// TIA Portal V20 export
FUNCTION_BLOCK "FB_ExtraMissingPart"   // FB76, SCL
{ S7_Optimized_Access := 'TRUE' }
// stored: MemoryReserve 100, SetENOAutomatically false
   VAR
      sRT_UndrilledGripperClosedWithPart : R_TRIG;
      sRT_UndrilledGripperClosedWithoutPart { S7_SetPoint := 'True'} : R_TRIG;
      sRT_DrilledGripperClosedWithPart : R_TRIG;
      sRT_DrilledGripperClosedWithoutPart { S7_SetPoint := 'True'} : R_TRIG;
      sRT_FixturePartControlGood { S7_SetPoint := 'True'} : R_TRIG;
      sRT_FixturePartControlBad { S7_SetPoint := 'True'} : R_TRIG;
      sRT_UndrilledGripperOpen { S7_SetPoint := 'True'} : R_TRIG;
      sRT_DrilledGripperOpen { S7_SetPoint := 'True'} : R_TRIG;
      sTON_UndrilledGripperClosedWithPart { S7_SetPoint := 'True'} : TON_TIME;
      sTON_UndrilledGripperClosedWithoutPart { S7_SetPoint := 'True'} : TON_TIME;
      sTON_DrilledGripperClosedWithPart { S7_SetPoint := 'True'} : TON_TIME;
      sTON_DrilledGripperClosedWithoutPart { S7_SetPoint := 'True'} : TON_TIME;
      sTON_FixturePartControlGood { S7_SetPoint := 'True'} : TON_TIME;
      sTON_FixturePartControlBad { S7_SetPoint := 'True'} : TON_TIME;
      sTON_UndrilledGripperOpen { S7_SetPoint := 'True'} : TON_TIME;
      sTON_DrilledGripperOpen { S7_SetPoint := 'True'} : TON_TIME;
      sExtraPartUndrilledGripper { S7_SetPoint := 'True'} : Bool;
      sExtraPartDrilledGripper : Bool;
      sMissingPartUndrilledGripper { S7_SetPoint := 'True'} : Bool;
      sMissingPartDrilledGripper : Bool;
      sExtraPartFixture : Bool;
      sMissingPartFixture : Bool;
      sGlobalExtraMissing : Bool;
      sUndrilledGripperClosedWithPart : Bool;
      sUndrilledGripperClosedWithoutPart { S7_SetPoint := 'True'} : Bool;
      sDrilledGripperClosedWithPart : Bool;
      sDrilledGripperClosedWithoutPart { S7_SetPoint := 'True'} : Bool;
      sFixturePartControlGood { S7_SetPoint := 'True'} : Bool;
      sFixturePartControlBad { S7_SetPoint := 'True'} : Bool;
      sUndrilledGripperOpen { S7_SetPoint := 'True'} : Bool;
      sDrilledGripperOpen { S7_SetPoint := 'True'} : Bool;
   END_VAR
BEGIN
   REGION Description header 
       //==================================================================================
       // POSALUX Swiss SA / (C) Copyright 2026
       //----------------------------------------------------------------------------------
       // Title: 
       // Comment/Function: 
       // Author: Fabien WALDT
       // Engineering: TIA Portal v20
       //----------------------------------------------------------------------------------
       // Change log table:
       // Version  | Date     | Expert in charge | Changes applied
       // ---------|----------|------------------|-----------------------------------------
       // 00.00.01 | 20260205 | WFA              | First released version
       // =================================================================================
   END_REGION

   REGION Init
       #sExtraPartUndrilledGripper := FALSE;
       #sExtraPartDrilledGripper := FALSE;
       #sMissingPartUndrilledGripper := FALSE;
       #sMissingPartDrilledGripper := FALSE;
       #sExtraPartFixture := FALSE;
       #sMissingPartFixture := FALSE;
   END_REGION

   REGION Inputs Status
       #sTON_UndrilledGripperClosedWithPart(IN := "DB_GestionGripper".sUndrilledGripper.oStateCloseWithPart,
                                            PT := T#100ms);
       #sTON_UndrilledGripperClosedWithoutPart(IN := "DB_GestionGripper".sUndrilledGripper.oStateClose,
                                               PT := T#100ms);
       #sTON_DrilledGripperClosedWithPart(IN := "DB_GestionGripper".sDrilledGripper.oStateCloseWithPart,
                                          PT := T#100ms);
       #sTON_DrilledGripperClosedWithoutPart(IN := "DB_GestionGripper".sDrilledGripper.oStateClose,
                                             PT := T#100ms);
       #sTON_FixturePartControlGood(IN := "DB_GestionFixture".sFixturePartControl.oGoodPart,
                                    PT := T#100ms);
       #sTON_FixturePartControlBad(IN := "DB_GestionFixture".sFixturePartControl.oBadpart,
                                   PT := T#100ms);

       #sTON_UndrilledGripperOpen(IN := "DB_GestionGripper".sUndrilledGripper.oStateOpen,
                                  PT := T#100ms);
       #sTON_DrilledGripperOpen(IN := "DB_GestionGripper".sDrilledGripper.oStateOpen,
                                PT := T#100ms);

       #sRT_UndrilledGripperClosedWithPart(CLK := #sTON_UndrilledGripperClosedWithPart.Q);
       #sRT_UndrilledGripperClosedWithoutPart(CLK := #sTON_UndrilledGripperClosedWithoutPart.Q);
       #sRT_DrilledGripperClosedWithPart(CLK := #sTON_DrilledGripperClosedWithPart.Q);
       #sRT_DrilledGripperClosedWithoutPart(CLK := #sTON_DrilledGripperClosedWithoutPart.Q);
       #sRT_FixturePartControlGood(CLK := #sTON_FixturePartControlGood.Q);
       #sRT_FixturePartControlBad(CLK := #sTON_FixturePartControlBad.Q);
       #sRT_UndrilledGripperOpen(CLK := #sTON_UndrilledGripperOpen.Q);
       #sRT_DrilledGripperOpen(CLK := #sTON_DrilledGripperOpen.Q);

       #sUndrilledGripperClosedWithPart := #sTON_UndrilledGripperClosedWithPart.Q;
       #sUndrilledGripperClosedWithoutPart := #sTON_UndrilledGripperClosedWithoutPart.Q;
       #sDrilledGripperClosedWithPart := #sTON_DrilledGripperClosedWithPart.Q;
       #sDrilledGripperClosedWithoutPart := #sTON_DrilledGripperClosedWithoutPart.Q;
       #sFixturePartControlGood := #sTON_FixturePartControlGood.Q;
       #sFixturePartControlBad := #sTON_FixturePartControlBad.Q;
       #sUndrilledGripperOpen := #sTON_UndrilledGripperOpen.Q;
       #sDrilledGripperOpen := #sTON_DrilledGripperOpen.Q;

   END_REGION

   REGION Shuttle to Undrilled Gripper
       IF "LBP_ModeGroup".E_JOG THEN
           IF #sRT_UndrilledGripperClosedWithPart.Q AND NOT "DB_PartManagement".sPosition.sGripper.Undrilled.Presence.Part THEN
               "DB_PartManagement".sPosition.sGripper.Undrilled.Presence.Part := TRUE;
               "DB_PartManagement".sPosition.sGripper.Undrilled.Presence.BW := TRUE;
           ELSIF #sRT_UndrilledGripperClosedWithoutPart.Q AND "DB_PartManagement".sPosition.sGripper.Undrilled.Presence.Part THEN
               "DB_PartManagement".sPosition.sGripper.Undrilled.Presence.Part := FALSE;
               "DB_PartManagement".sPosition.sGripper.Undrilled.Presence.BW := FALSE;
           END_IF;
       ELSIF NOT "DB_WorkingModes".sDryRun THEN
           IF #sUndrilledGripperClosedWithPart AND NOT "DB_PartManagement".sPosition.sGripper.Undrilled.Presence.Part THEN
               #sExtraPartUndrilledGripper := TRUE;
               "LBP_AlarmMsgs".UserA[04].A70UUxx[25] := TRUE; // Msg 700425 "Extra Product Undrilled Gripper"
           ELSIF #sUndrilledGripperClosedWithoutPart AND "DB_PartManagement".sPosition.sGripper.Undrilled.Presence.Part THEN
               #sMissingPartUndrilledGripper := TRUE;
               "LBP_AlarmMsgs".UserA[04].A70UUxx[24] := TRUE; // Msg 700424 "Missing Product Undrilled Gripper"
           END_IF;
       END_IF;
   END_REGION

   REGION Undrilled Gripper to Fixture
       IF "LBP_ModeGroup".E_JOG THEN
           IF #sRT_FixturePartControlGood.Q AND NOT "DB_PartManagement".sPosition.sFixture.Undrilled.Presence.Part AND NOT "DB_PartManagement".sPosition.sFixture.Drilled.Presence.Part THEN
               "DB_PartManagement".sPosition.sFixture.Drilled.Presence.Part := TRUE;
               "DB_PartManagement".sPosition.sFixture.Drilled.Presence.BW := TRUE;
           ELSIF #sRT_FixturePartControlBad.Q AND ("DB_PartManagement".sPosition.sFixture.Undrilled.Presence.Part OR "DB_PartManagement".sPosition.sFixture.Drilled.Presence.Part) THEN
               "DB_PartManagement".sPosition.sFixture.Drilled.Presence.Part := FALSE;
               "DB_PartManagement".sPosition.sFixture.Drilled.Presence.BW := FALSE;
           END_IF;
       ELSIF NOT "DB_WorkingModes".sDryRun THEN
           IF #sFixturePartControlGood AND NOT "DB_PartManagement".sPosition.sFixture.Undrilled.Presence.Part AND NOT "DB_PartManagement".sPosition.sFixture.Drilled.Presence.Part THEN
               #sExtraPartFixture := TRUE;
               "LBP_AlarmMsgs".UserA[04].A70UUxx[27] := TRUE; // Msg 700427 "Extra Product Fixture"
           ELSIF #sFixturePartControlBad AND ("DB_PartManagement".sPosition.sFixture.Undrilled.Presence.Part OR "DB_PartManagement".sPosition.sFixture.Drilled.Presence.Part) THEN
               #sMissingPartFixture := TRUE;
               "LBP_AlarmMsgs".UserA[04].A70UUxx[26] := TRUE; // Msg 700426 "Missing Product Fixture"
           END_IF;
       END_IF;
   END_REGION

   REGION Fixture to Drilled Gripper
       IF "LBP_ModeGroup".E_JOG THEN
           IF #sRT_DrilledGripperClosedWithPart.Q AND NOT "DB_PartManagement".sPosition.sGripper.Drilled.Presence.Part THEN
               "DB_PartManagement".sPosition.sGripper.Drilled.Presence.Part := TRUE;
               "DB_PartManagement".sPosition.sGripper.Drilled.Presence.BW := TRUE;
           ELSIF #sRT_DrilledGripperClosedWithoutPart.Q AND "DB_PartManagement".sPosition.sGripper.Drilled.Presence.Part THEN
               "DB_PartManagement".sPosition.sGripper.Drilled.Presence.Part := FALSE;
               "DB_PartManagement".sPosition.sGripper.Drilled.Presence.BW := FALSE;
           END_IF;
       ELSIF NOT "DB_WorkingModes".sDryRun THEN
           IF #sDrilledGripperClosedWithPart AND NOT "DB_PartManagement".sPosition.sGripper.Drilled.Presence.Part THEN
               #sExtraPartDrilledGripper := TRUE;
               "LBP_AlarmMsgs".UserA[04].A70UUxx[29] := TRUE; // Msg 700429 "Extra Product Drilled Gripper"
           ELSIF #sDrilledGripperClosedWithoutPart AND "DB_PartManagement".sPosition.sGripper.Drilled.Presence.Part THEN
               #sMissingPartDrilledGripper := TRUE;
               "LBP_AlarmMsgs".UserA[04].A70UUxx[28] := TRUE; // Msg 700428 "Missing Product Drilled Gripper"
           END_IF;
       END_IF;
   END_REGION

   REGION Gripper Open
       IF "LBP_ModeGroup".E_JOG THEN
           IF #sRT_UndrilledGripperOpen.Q THEN
               "DB_PartManagement".sPosition.sGripper.Undrilled.Presence.Part := FALSE;
               "DB_PartManagement".sPosition.sGripper.Undrilled.Presence.BW := FALSE;
           END_IF;
           IF #sRT_DrilledGripperOpen.Q THEN
               "DB_PartManagement".sPosition.sGripper.Drilled.Presence.Part := FALSE;
               "DB_PartManagement".sPosition.sGripper.Drilled.Presence.BW := FALSE;
           END_IF;
       END_IF;
   END_REGION

   REGION Global Extra Missing
       #sGlobalExtraMissing :=
          #sExtraPartUndrilledGripper
       OR #sExtraPartDrilledGripper
       OR #sMissingPartUndrilledGripper 
       OR #sMissingPartDrilledGripper
       OR #sExtraPartFixture
       OR #sMissingPartFixture;
   END_REGION
END_FUNCTION_BLOCK
